// TIA Portal V20 export
TYPE "s_zc_IntercellSafetyDeviceToAdjCell"
// stored: Access Published, IsFailsafeCompliant true, Namespace Safety
   STRUCT
      SDConnected { ExternalWritable := 'False'} : Bool := FALSE;   // Safety Device(s) Connected
      SDClear { ExternalWritable := 'False'} : Bool := FALSE;   // Safety Device(s) Clear
      OtherSDsOK { ExternalWritable := 'False'} : Bool := FALSE;   // All Other Safety Devices OK
      OutsideGateReset { ExternalWritable := 'False'} : Bool := FALSE;   // Outside Gates Reset
      PendantActivated { ExternalWritable := 'False'} : Bool := FALSE;   // Pendant HMI is connected and actvated to use via Enable button.
      MPSActivated { ExternalWritable := 'False'} : Bool := FALSE;   // All safety output devices and motions are deenergized and they are monitored by safety feedback.
      EnableMotion { ExternalWritable := 'False'} : Bool := FALSE;   // Enable Equipment Within 1.5 meters of Intercell
      EnableWarning { ExternalWritable := 'False'} : Bool := FALSE;   // Enabl Timer Running Hold Adj Equipment
      ResetSDReq { ExternalWritable := 'False'} : Bool := FALSE;   // Reset PB Pressed
      ResetLightFlash { ExternalWritable := 'False'} : Bool := FALSE;   // Flash Reset Light
      ResetLightSolid { ExternalWritable := 'False'} : Bool := FALSE;   // Turn On Reset Light
      LoadingProtectionAreaOK { ExternalWritable := 'False'} : Bool := FALSE;   // Loading area is protected and loader/gantry can traverse in load area.
      EnableOpenSafetyGate { ExternalWritable := 'False'} : Bool := FALSE;   // Machine is stopped, so operator can open the safety gate.
   END_STRUCT;
END_TYPE
